// TIA Portal V16 export
// export: Created 2021-09-08T12:46:11.4713699Z, ExportSetting WithDefaults, DisplayName Totally Integrated Automation Portal, DisplayVersion V16 Update 3, DisplayName TIA Portal Version Control Interface, DisplayVersion V16 Update 2, DisplayName TIA Portal Openness, DisplayVersion V16 Update 3, DisplayName TIA Portal Teamcenter Gateway, DisplayVersion V16, DisplayName STEP 7 Professional, DisplayVersion V16 Update 3, DisplayName STEP 7 Safety, DisplayVersion V16, DisplayName WinCC Advanced, DisplayVersion V16 Update 3
FUNCTION_BLOCK "sel2pu"   // FB4, FBD
{ S7_Optimized_Access := 'TRUE' }
VERSION : 0.1
// stored: AutoNumber true, IsIECCheckEnabled false, IsRetainMemResEnabled false, MemoryReserve 100, SetENOAutomatically false, UDAEnableTagReadback false
   VAR_INPUT
      cmStart : Bool;
      mode : Bool;
      tChangeHReal : Real;
   END_VAR
   VAR_OUTPUT
      tToChange : Real;
   END_VAR
   VAR_IN_OUT
      PU1 : "Pump";
      PU2 : "Pump";
      select : Bool;
   END_VAR
   VAR
      tWork1 : DInt;
      tWork2 : DInt;
      tChangeDInt : DInt;
   END_VAR
BEGIN

REGION Network 1: Режим работы
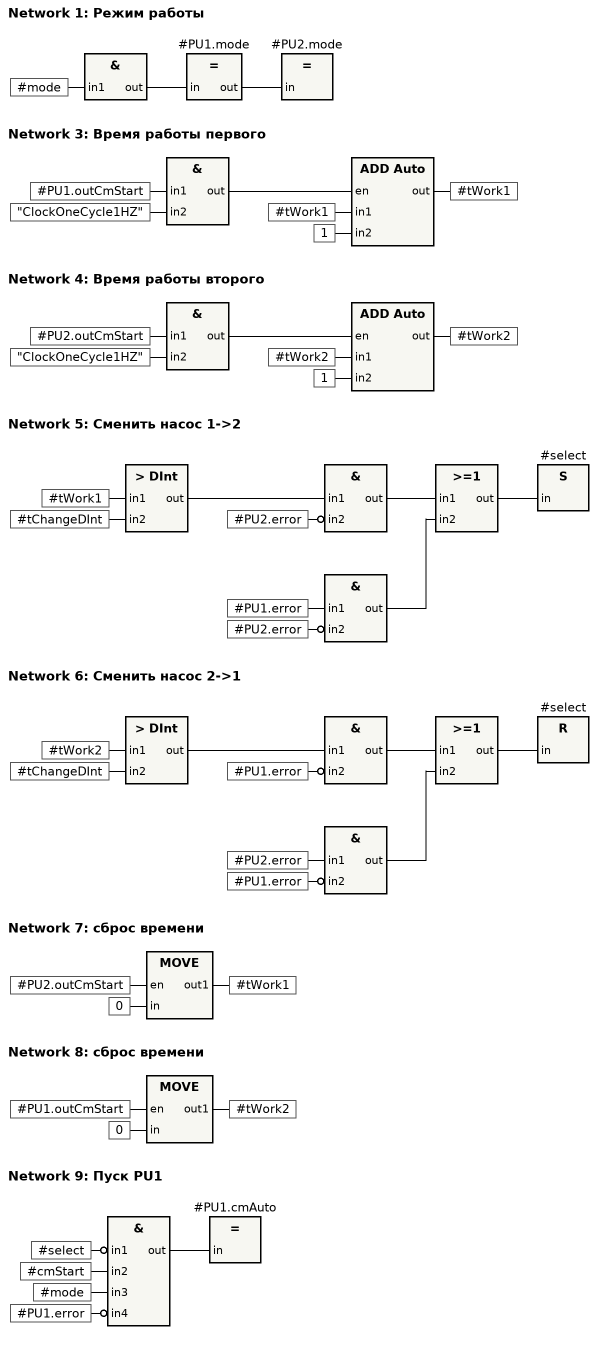
   #PU1.mode := #mode;
   #PU2.mode := #mode;
END_REGION

REGION Network 2 (SCL): Преобразование времен
   #tChangeDInt := REAL_TO_DINT(#tChangeHReal * 3600.0);
END_REGION

REGION Network 3: Время работы первого
   IF #PU1.outCmStart AND "ClockOneCycle1HZ" THEN #tWork1 := #tWork1 + 1; END_IF;
END_REGION

REGION Network 4: Время работы второго
   IF #PU2.outCmStart AND "ClockOneCycle1HZ" THEN #tWork2 := #tWork2 + 1; END_IF;
END_REGION

REGION Network 5: Сменить насос 1->2
   IF ((#tWork1 > #tChangeDInt) AND NOT #PU2.error) OR (#PU1.error AND NOT #PU2.error) THEN
       #select := TRUE;
   END_IF;
END_REGION

REGION Network 6: Сменить насос 2->1
   IF ((#tWork2 > #tChangeDInt) AND NOT #PU1.error) OR (#PU2.error AND NOT #PU1.error) THEN
       #select := FALSE;
   END_IF;
END_REGION

REGION Network 7: сброс времени
   IF #PU2.outCmStart THEN #tWork1 := 0; END_IF;
END_REGION

REGION Network 8: сброс времени
   IF #PU1.outCmStart THEN #tWork2 := 0; END_IF;
END_REGION

REGION Network 9: Пуск PU1
   #PU1.cmAuto := NOT #select AND #cmStart AND #mode AND NOT #PU1.error;
END_REGION

REGION Network 10: Пуск PU2
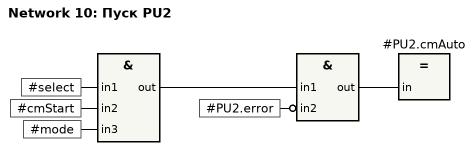
   #PU2.cmAuto := #select AND #cmStart AND #mode AND NOT #PU2.error;
END_REGION
END_FUNCTION_BLOCK
